// TwinCAT 3 PLC project plc_project
// ProgramVersion: 3.1.4024.0
// libraries:
//   Tc2_Standard, * (Beckhoff Automation GmbH)
//   Tc2_System, * (Beckhoff Automation GmbH)
//   Tc3_Module, * (Beckhoff Automation GmbH)
// project tree:
//   GVLs/ GVL.TcGVL
//   / PlcTask1.TcTTO, PlcTask2.TcTTO
//   POUs/ program1.TcPOU, program2.TcPOU
// real-time tasks:
//   TASK PlcTask1: cycle T#10ms, priority 1, ADS port 350
//   TASK PlcTask2: cycle T#10ms, priority 2, ADS port 351

CONFIGURATION plc_project
    RESOURCE PLC ON TwinCAT3
        TASK PlcTask1(INTERVAL := T#10ms, PRIORITY := 1);
        TASK PlcTask2(INTERVAL := T#10ms, PRIORITY := 2);
        PROGRAM program1 WITH PlcTask1 : program1;
        PROGRAM program2 WITH PlcTask2 : program2;
    END_RESOURCE
END_CONFIGURATION

// ---- GVLs/GVL.TcGVL
{attribute 'qualified_only'}
VAR_GLOBAL
END_VAR

// ---- POUs/program1.TcPOU
PROGRAM program1
VAR
	to_2 : INT := 0;
	from_2 : INT := 0;
END_VAR

gvl.from_1_to_2 := to_2;
from_2 := gvl.from_2_to_1;

END_PROGRAM

// ---- POUs/program2.TcPOU
PROGRAM program2
VAR
	to_1 : INT := 0;
	from_1 : INT := 0;
END_VAR

from_1 := gvl.from_1_to_2;
to_1 := from_1 + 10;
gvl.from_2_to_1 := to_1;

END_PROGRAM
